TYPE TPearlingTeachPos :
	(
		PTP_TableSideAPosZ1 := 0,
		PTP_TableSideAPosZ2,
		PTP_TableSideBPosZ1,
		PTP_TableSideBPosZ2,
		PTP_BarrelPosZ1,
		PTP_BarrelPosZ2,
		PTP_RejectPosZ1,
		PTP_RejectPosZ2,
		PTP_Sharpen,
		PTP_WeightCalibrationPosZ1,
		PTP_WeightCalibrationPosZ2,
		PTP_END
	);
END_TYPE

(* stored: Version 1.1.0.1, ProductVersion 3.1.4022.12
   DUT TPearlingTeachPos: Id {b9947de1-ae59-4b4f-a721-307a9821bdeb} *)
